// TIA Portal V19 export
TYPE "FeedMachine_DataOut"
// stored: Access Published
   STRUCT
      Fan_M_Contactor : Bool;
   END_STRUCT;
END_TYPE
